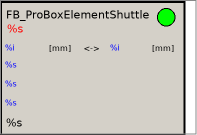
VISUALIZATION V_Element_Shuttle  // 197x135
VAR_IN_OUT
	{attribute 'VAR_IN_OUT_AS_POINTER'}
	fbFunction		: FB_ProBoxElementShuttle;
	//fbEmuFunction	: FB_ProBOXSG_Emulation;
END_VAR
    Rectangle (0,1 185x134), colour toggle: fbFunction.fbMpdControl.CtrlOut.MotionRunning
    Rectangle (3,113 143x20), "%s", text variable: fbFunction.ConfigElement.ElementName
    Label (3,5 158x20), "FB_ProBoxElementShuttle"
    Rectangle (2,38 54x20), "%i", tooltip "'Actual driver positon'", text variable: fbFunction.fbMpdControl._MPD.ActualPosValue
    Rectangle (4,19 161x20), "%s", tooltip "%s", text variable: fbFunction.ElementData.ErrorData.Error.ErrorCode.Conv, invisible if: fbFunction.ElementData.ErrorData.Error.ErrorCode.Conv = 0
        p4168582468: fbFunction.ElementData.ErrorData.Error.ErrorParam
    Rectangle (107,38 58x20), "%i", tooltip "'Set position'", text variable: fbFunction.fbMpdControl._MPD.RequestPosValue
        p4168582468: 'Set Position'
    Ellipse (157,8 18x18), colour toggle: NOT fbFunction.HW_Inputs.MotorUnitOK
    Label (45,42 30x13), "[mm]"
    Label (77,42 29x13), "<->"
    Rectangle (2,55 127x20), "%s", tooltip "'MPD State'", text variable: fbFunction.fbMpdControl._MPD.State
    Rectangle (2,74 195x20), "%s", text variable: fbFunction.fbMpdControl._MPD.CV[1].PickupFuncNumber
        p4168582468: 'PickupFuncNumber'
    Rectangle (2,93 183x20), "%s", text variable: fbFunction.fbMpdControl._MPD.CV[1].DepositFuncNumber
        p4168582468: 'DepositFuncNumber'
    Label (148,42 30x13), "[mm]"
END_VISUALIZATION

(* stored: Version 1.1.0.1, ProductVersion 3.1.4024.9
   Visu V_Element_Shuttle: Id {6a66b5a2-fe56-4bcb-8893-d2c69a83bbb0} *)
